(* Logix 5000 project; controller Generic 1768-L43 rev 16.2; software revision 15.01; part 5 of 10 *)
(* tags used below, declared in another part *)
   EL_CTRL_1 : UDT_AxisHistory_CTRL;
   EL_CTRL_2 : UDT_AxisHistory_CTRL;
   EL_CTRL_3 : UDT_AxisHistory_CTRL;
   EL_CTRL_4 : UDT_AxisHistory_CTRL;
   EL_CTRL_5 : UDT_AxisHistory_CTRL;
   EL_CTRL_6 : UDT_AxisHistory_CTRL;
   EL_CTRL_7 : UDT_AxisHistory_CTRL;
   EL_CTRL_8 : UDT_AxisHistory_CTRL;
   EL_SaveSEQ : DINT;
   EventINDEX : DINT;
   EventLog_N1 : UDT_AxisHistory_DLM[51];
   EventLog_N2 : UDT_AxisHistory_DLM[51];
   EventLog_N3 : UDT_AxisHistory_DLM[51];
   EventLog_N4 : UDT_AxisHistory_DLM[51];
   EventLog_N5 : UDT_AxisHistory_DLM[51];
   EventLog_N6 : UDT_AxisHistory_DLM[51];
   EventLog_N7 : UDT_AxisHistory_DLM[51];
   EventLog_N8 : UDT_AxisHistory_DLM[51];
   GUI_DataDisplay : UDT_AxisHistory_DLM;
   GUI_DataLogModel : UDT_AxisHistory_DLM;
   GUI_EventLogSaving : BOOL;
   GUI_IndexSelect : DINT;
   GUI_NodeSelect : DINT;
   GUI_SaveEventLog : BOOL;
   LogLength : DINT;
   PowerUP_TMR : TIMER;
   Axis_00_Data : UDT_Axis_Data;
   Axis_00_Status : UDT_Axis_Status;
   AXIS_01 : AXIS_SERVO_DRIVE;
   Axis_01_Data : UDT_Axis_Data;
   Axis_01_Status : UDT_Axis_Status;
   AXIS_02 : AXIS_SERVO_DRIVE;
   Axis_02_Data : UDT_Axis_Data;
   Axis_02_Status : UDT_Axis_Status;
   AXIS_03 : AXIS_SERVO_DRIVE;
   Axis_03_Data : UDT_Axis_Data;
   Axis_03_Status : UDT_Axis_Status;
   AXIS_04 : AXIS_SERVO_DRIVE;
   Axis_04_Data : UDT_Axis_Data;
   Axis_04_Status : UDT_Axis_Status;
   C_pi : REAL;
   GenericMachine_COND : UDT_Machine_COND;
   MASK : DINT;
(* AXIS_EventLog, continued *)

ROUTINE R20_HMI_EventLog   (* ladder *)
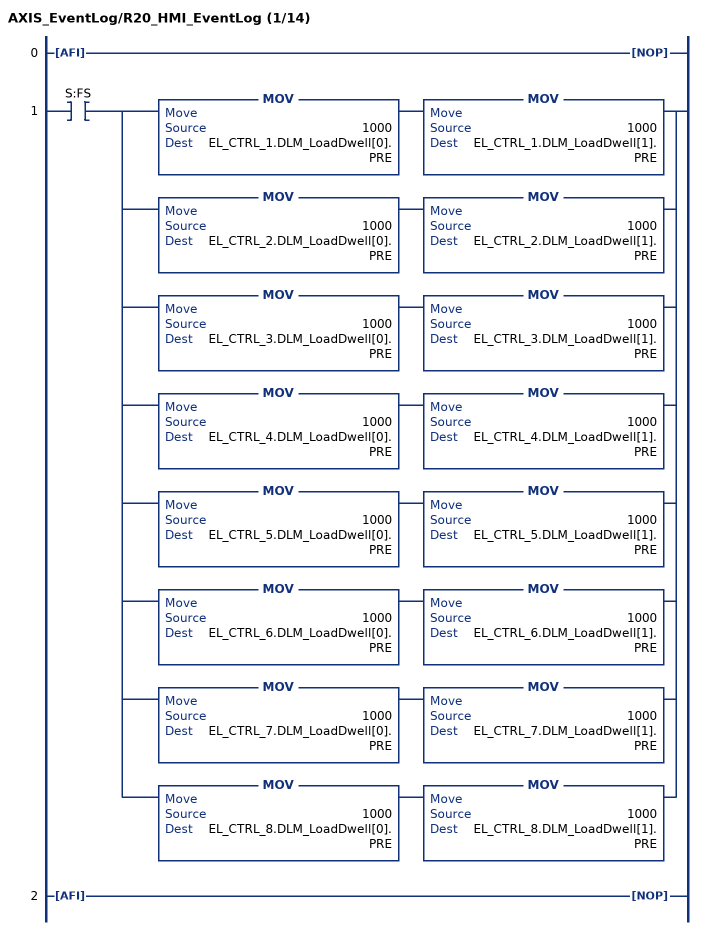
   0: AFI()NOP();
   1: XIC(S:FS)[MOV(1000,EL_CTRL_1.DLM_LoadDwell[0].PRE) MOV(1000,EL_CTRL_1.DLM_LoadDwell[1].PRE) ,MOV(1000,EL_CTRL_2.DLM_LoadDwell[0].PRE) MOV(1000,EL_CTRL_2.DLM_LoadDwell[1].PRE) ,MOV(1000,EL_CTRL_3.DLM_LoadDwell[0].PRE) MOV(1000,EL_CTRL_3.DLM_LoadDwell[1].PRE) ,MOV(1000,EL_CTRL_4.DLM_LoadDwell[0].PRE) MOV(1000,EL_CTRL_4.DLM_LoadDwell[1].PRE) ,MOV(1000,EL_CTRL_5.DLM_LoadDwell[0].PRE) MOV(1000,EL_CTRL_5.DLM_LoadDwell[1].PRE) ,MOV(1000,EL_CTRL_6.DLM_LoadDwell[0].PRE) MOV(1000,EL_CTRL_6.DLM_LoadDwell[1].PRE) ,MOV(1000,EL_CTRL_7.DLM_LoadDwell[0].PRE) MOV(1000,EL_CTRL_7.DLM_LoadDwell[1].PRE) ,MOV(1000,EL_CTRL_8.DLM_LoadDwell[0].PRE) MOV(1000,EL_CTRL_8.DLM_LoadDwell[1].PRE) ];
   2: AFI()NOP();
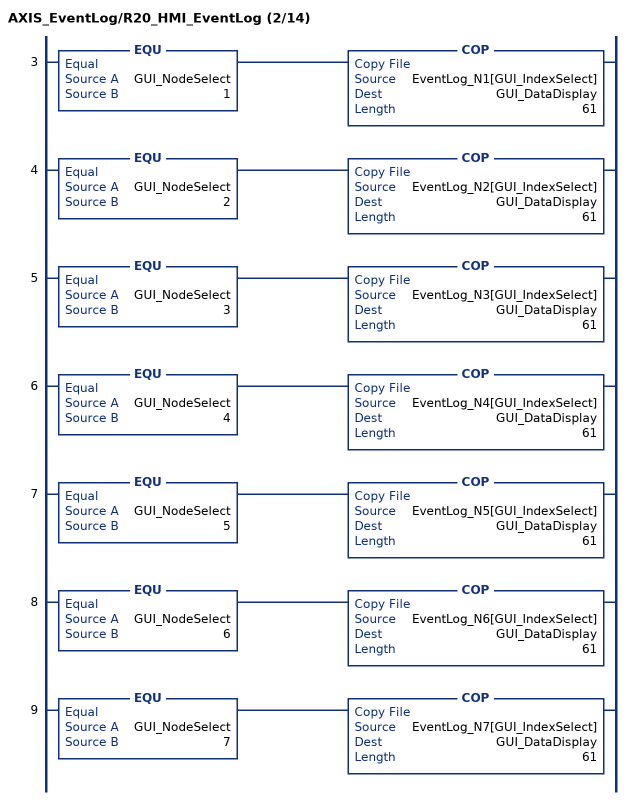
   3: EQU(GUI_NodeSelect,1)COP(EventLog_N1[GUI_IndexSelect],GUI_DataDisplay,61);
   4: EQU(GUI_NodeSelect,2)COP(EventLog_N2[GUI_IndexSelect],GUI_DataDisplay,61);
   5: EQU(GUI_NodeSelect,3)COP(EventLog_N3[GUI_IndexSelect],GUI_DataDisplay,61);
   6: EQU(GUI_NodeSelect,4)COP(EventLog_N4[GUI_IndexSelect],GUI_DataDisplay,61);
   7: EQU(GUI_NodeSelect,5)COP(EventLog_N5[GUI_IndexSelect],GUI_DataDisplay,61);
   8: EQU(GUI_NodeSelect,6)COP(EventLog_N6[GUI_IndexSelect],GUI_DataDisplay,61);
   9: EQU(GUI_NodeSelect,7)COP(EventLog_N7[GUI_IndexSelect],GUI_DataDisplay,61);
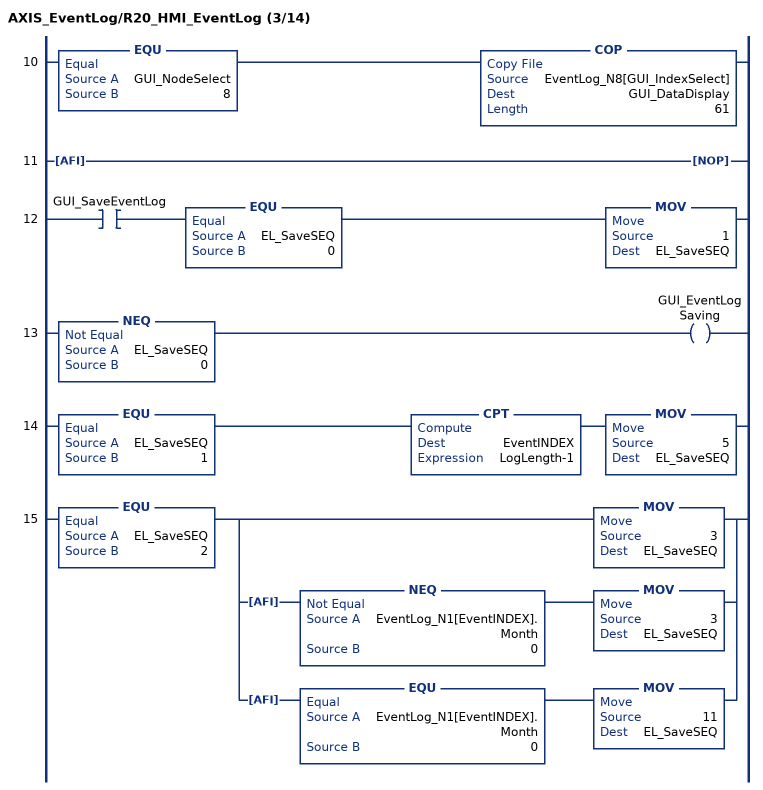
   10: EQU(GUI_NodeSelect,8)COP(EventLog_N8[GUI_IndexSelect],GUI_DataDisplay,61);
   11: AFI()NOP();
   12: XIC(GUI_SaveEventLog)EQU(EL_SaveSEQ,0)MOV(1,EL_SaveSEQ);
   13: NEQ(EL_SaveSEQ,0)OTE(GUI_EventLogSaving);
   14: EQU(EL_SaveSEQ,1)CPT(EventINDEX,LogLength-1)MOV(5,EL_SaveSEQ);
   15: EQU(EL_SaveSEQ,2)[MOV(3,EL_SaveSEQ) ,AFI() NEQ(EventLog_N1[EventINDEX].Month,0) MOV(3,EL_SaveSEQ) ,AFI() EQU(EventLog_N1[EventINDEX].Month,0) MOV(11,EL_SaveSEQ) ];
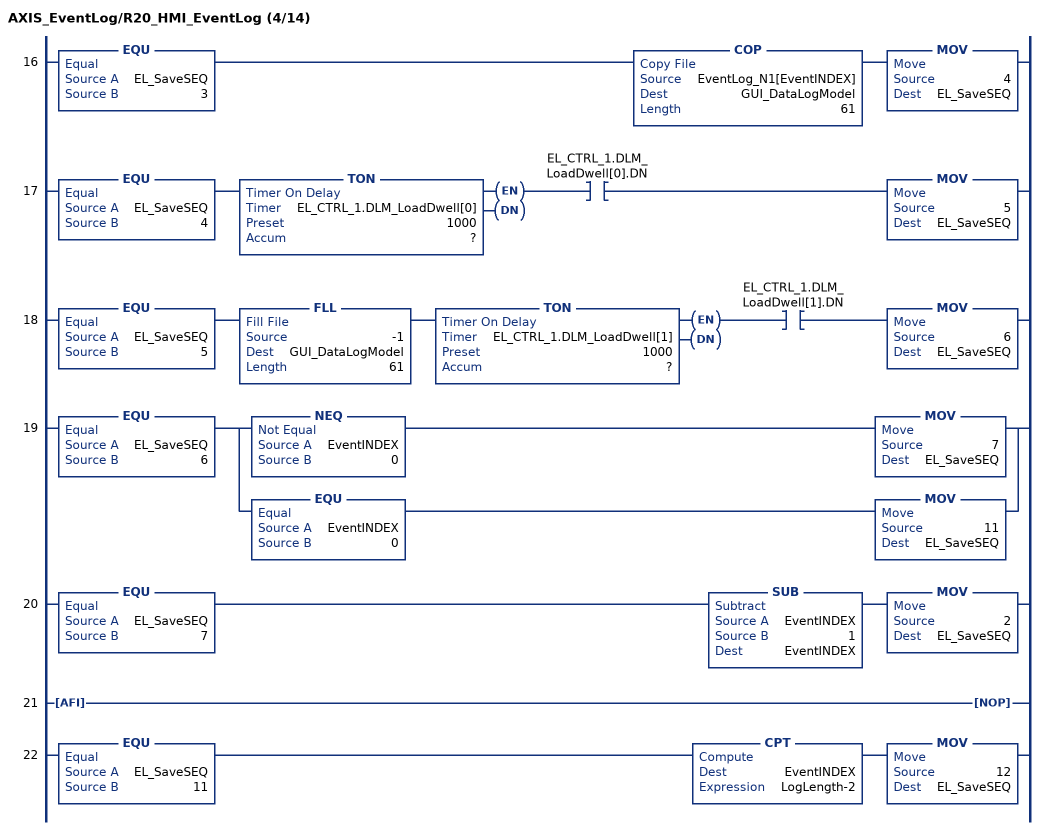
   16: EQU(EL_SaveSEQ,3)COP(EventLog_N1[EventINDEX],GUI_DataLogModel,61)MOV(4,EL_SaveSEQ);
   17: EQU(EL_SaveSEQ,4)TON(EL_CTRL_1.DLM_LoadDwell[0],?,?)XIC(EL_CTRL_1.DLM_LoadDwell[0].DN)MOV(5,EL_SaveSEQ);
   18: EQU(EL_SaveSEQ,5)FLL(-1,GUI_DataLogModel,61)TON(EL_CTRL_1.DLM_LoadDwell[1],?,?)XIC(EL_CTRL_1.DLM_LoadDwell[1].DN)MOV(6,EL_SaveSEQ);
   19: EQU(EL_SaveSEQ,6)[NEQ(EventINDEX,0) MOV(7,EL_SaveSEQ) ,EQU(EventINDEX,0) MOV(11,EL_SaveSEQ) ];
   20: EQU(EL_SaveSEQ,7)SUB(EventINDEX,1,EventINDEX)MOV(2,EL_SaveSEQ);
   21: AFI()NOP();
   22: EQU(EL_SaveSEQ,11)CPT(EventINDEX,LogLength-2)MOV(12,EL_SaveSEQ);
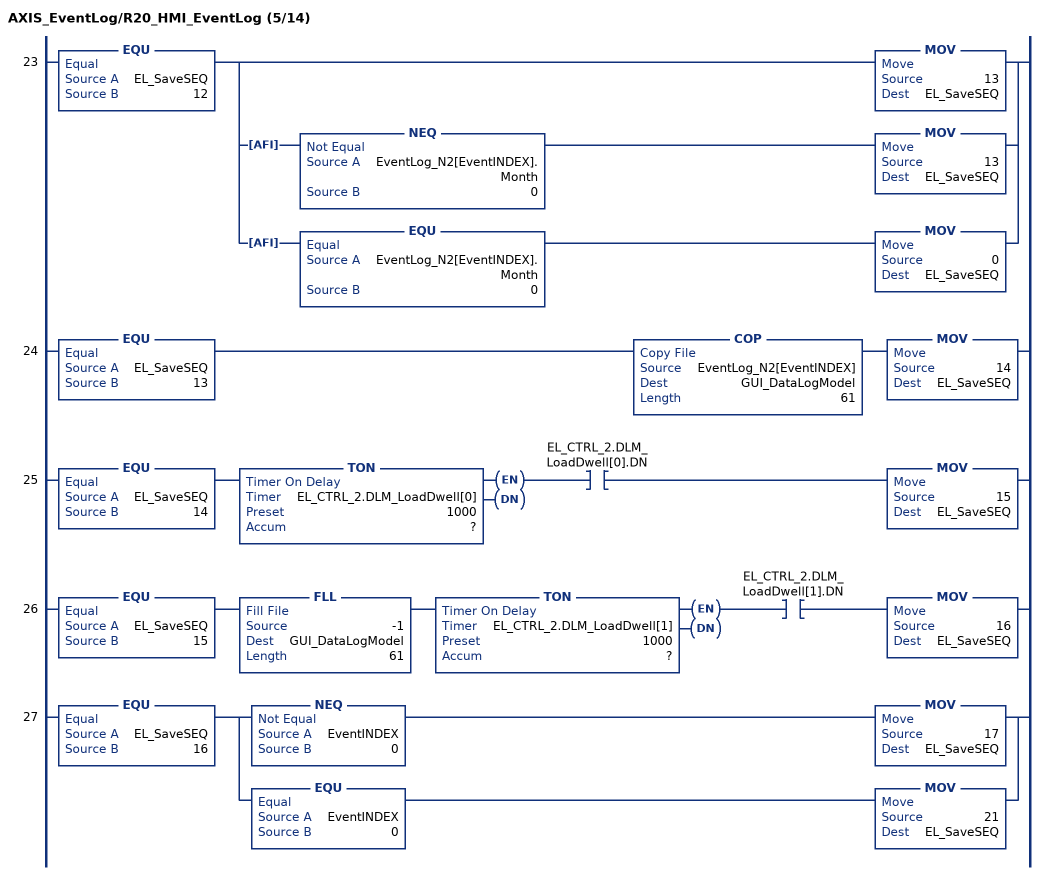
   23: EQU(EL_SaveSEQ,12)[MOV(13,EL_SaveSEQ) ,AFI() NEQ(EventLog_N2[EventINDEX].Month,0) MOV(13,EL_SaveSEQ) ,AFI() EQU(EventLog_N2[EventINDEX].Month,0) MOV(0,EL_SaveSEQ) ];
   24: EQU(EL_SaveSEQ,13)COP(EventLog_N2[EventINDEX],GUI_DataLogModel,61)MOV(14,EL_SaveSEQ);
   25: EQU(EL_SaveSEQ,14)TON(EL_CTRL_2.DLM_LoadDwell[0],?,?)XIC(EL_CTRL_2.DLM_LoadDwell[0].DN)MOV(15,EL_SaveSEQ);
   26: EQU(EL_SaveSEQ,15)FLL(-1,GUI_DataLogModel,61)TON(EL_CTRL_2.DLM_LoadDwell[1],?,?)XIC(EL_CTRL_2.DLM_LoadDwell[1].DN)MOV(16,EL_SaveSEQ);
   27: EQU(EL_SaveSEQ,16)[NEQ(EventINDEX,0) MOV(17,EL_SaveSEQ) ,EQU(EventINDEX,0) MOV(21,EL_SaveSEQ) ];
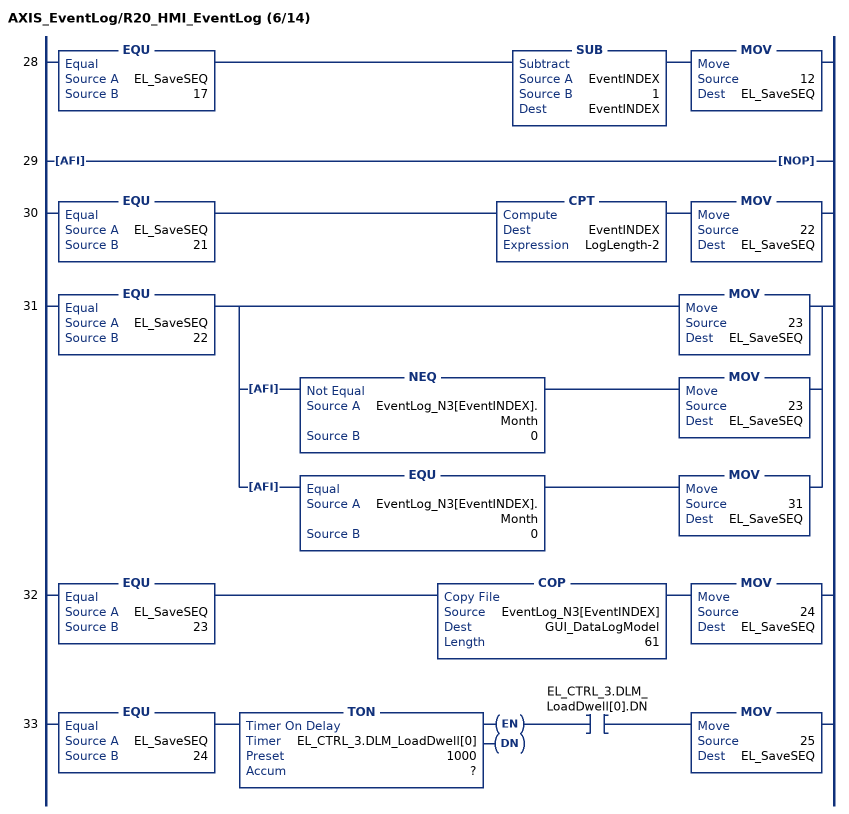
   28: EQU(EL_SaveSEQ,17)SUB(EventINDEX,1,EventINDEX)MOV(12,EL_SaveSEQ);
   29: AFI()NOP();
   30: EQU(EL_SaveSEQ,21)CPT(EventINDEX,LogLength-2)MOV(22,EL_SaveSEQ);
   31: EQU(EL_SaveSEQ,22)[MOV(23,EL_SaveSEQ) ,AFI() NEQ(EventLog_N3[EventINDEX].Month,0) MOV(23,EL_SaveSEQ) ,AFI() EQU(EventLog_N3[EventINDEX].Month,0) MOV(31,EL_SaveSEQ) ];
   32: EQU(EL_SaveSEQ,23)COP(EventLog_N3[EventINDEX],GUI_DataLogModel,61)MOV(24,EL_SaveSEQ);
   33: EQU(EL_SaveSEQ,24)TON(EL_CTRL_3.DLM_LoadDwell[0],?,?)XIC(EL_CTRL_3.DLM_LoadDwell[0].DN)MOV(25,EL_SaveSEQ);
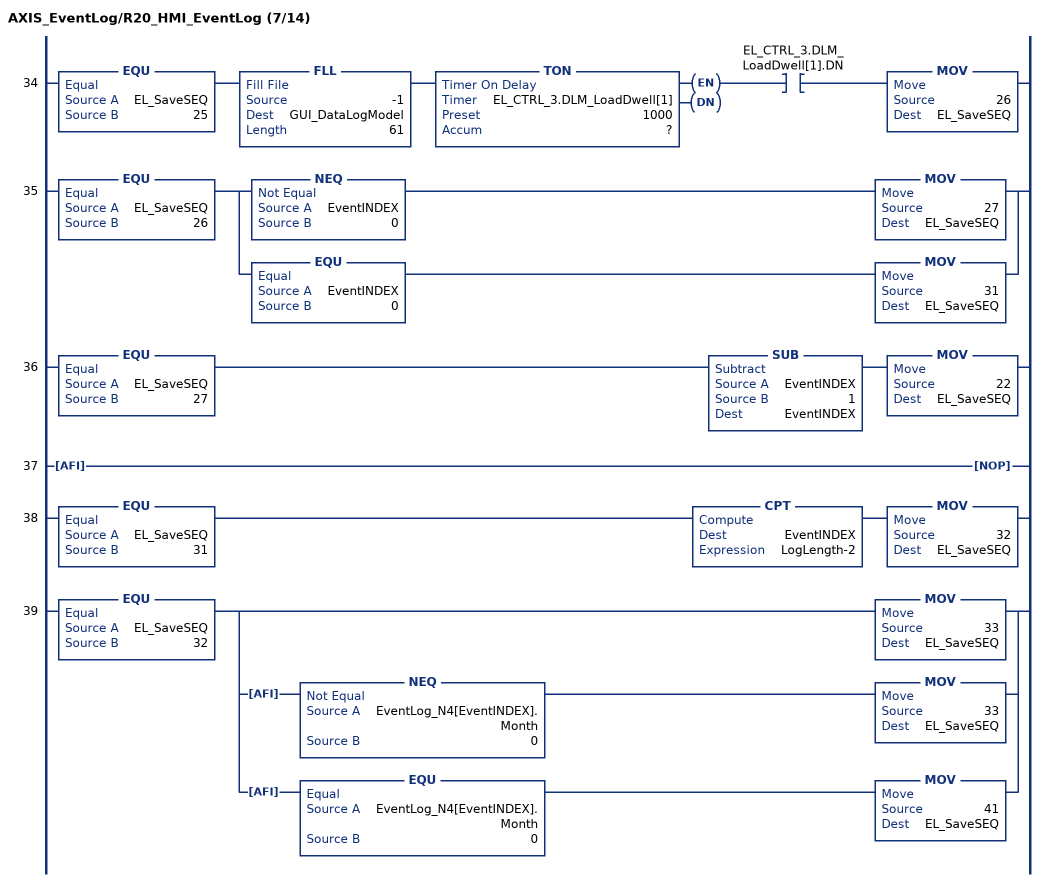
   34: EQU(EL_SaveSEQ,25)FLL(-1,GUI_DataLogModel,61)TON(EL_CTRL_3.DLM_LoadDwell[1],?,?)XIC(EL_CTRL_3.DLM_LoadDwell[1].DN)MOV(26,EL_SaveSEQ);
   35: EQU(EL_SaveSEQ,26)[NEQ(EventINDEX,0) MOV(27,EL_SaveSEQ) ,EQU(EventINDEX,0) MOV(31,EL_SaveSEQ) ];
   36: EQU(EL_SaveSEQ,27)SUB(EventINDEX,1,EventINDEX)MOV(22,EL_SaveSEQ);
   37: AFI()NOP();
   38: EQU(EL_SaveSEQ,31)CPT(EventINDEX,LogLength-2)MOV(32,EL_SaveSEQ);
   39: EQU(EL_SaveSEQ,32)[MOV(33,EL_SaveSEQ) ,AFI() NEQ(EventLog_N4[EventINDEX].Month,0) MOV(33,EL_SaveSEQ) ,AFI() EQU(EventLog_N4[EventINDEX].Month,0) MOV(41,EL_SaveSEQ) ];
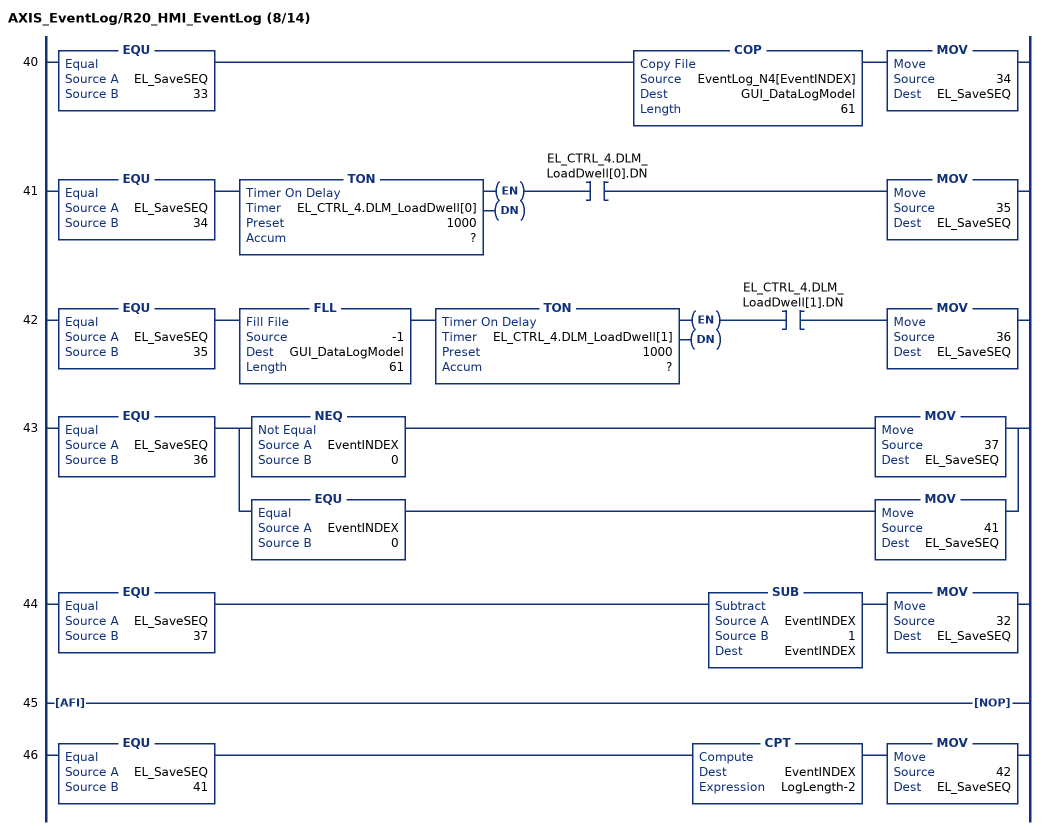
   40: EQU(EL_SaveSEQ,33)COP(EventLog_N4[EventINDEX],GUI_DataLogModel,61)MOV(34,EL_SaveSEQ);
   41: EQU(EL_SaveSEQ,34)TON(EL_CTRL_4.DLM_LoadDwell[0],?,?)XIC(EL_CTRL_4.DLM_LoadDwell[0].DN)MOV(35,EL_SaveSEQ);
   42: EQU(EL_SaveSEQ,35)FLL(-1,GUI_DataLogModel,61)TON(EL_CTRL_4.DLM_LoadDwell[1],?,?)XIC(EL_CTRL_4.DLM_LoadDwell[1].DN)MOV(36,EL_SaveSEQ);
   43: EQU(EL_SaveSEQ,36)[NEQ(EventINDEX,0) MOV(37,EL_SaveSEQ) ,EQU(EventINDEX,0) MOV(41,EL_SaveSEQ) ];
   44: EQU(EL_SaveSEQ,37)SUB(EventINDEX,1,EventINDEX)MOV(32,EL_SaveSEQ);
   45: AFI()NOP();
   46: EQU(EL_SaveSEQ,41)CPT(EventINDEX,LogLength-2)MOV(42,EL_SaveSEQ);
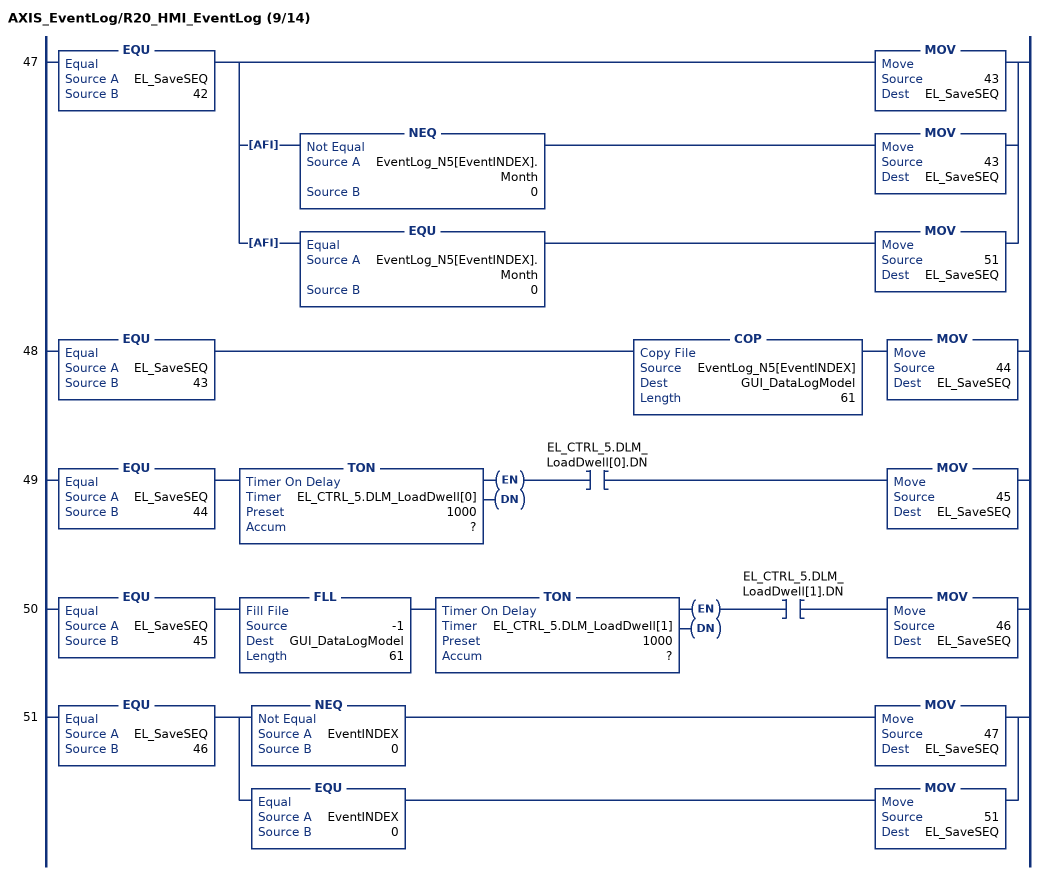
   47: EQU(EL_SaveSEQ,42)[MOV(43,EL_SaveSEQ) ,AFI() NEQ(EventLog_N5[EventINDEX].Month,0) MOV(43,EL_SaveSEQ) ,AFI() EQU(EventLog_N5[EventINDEX].Month,0) MOV(51,EL_SaveSEQ) ];
   48: EQU(EL_SaveSEQ,43)COP(EventLog_N5[EventINDEX],GUI_DataLogModel,61)MOV(44,EL_SaveSEQ);
   49: EQU(EL_SaveSEQ,44)TON(EL_CTRL_5.DLM_LoadDwell[0],?,?)XIC(EL_CTRL_5.DLM_LoadDwell[0].DN)MOV(45,EL_SaveSEQ);
   50: EQU(EL_SaveSEQ,45)FLL(-1,GUI_DataLogModel,61)TON(EL_CTRL_5.DLM_LoadDwell[1],?,?)XIC(EL_CTRL_5.DLM_LoadDwell[1].DN)MOV(46,EL_SaveSEQ);
   51: EQU(EL_SaveSEQ,46)[NEQ(EventINDEX,0) MOV(47,EL_SaveSEQ) ,EQU(EventINDEX,0) MOV(51,EL_SaveSEQ) ];
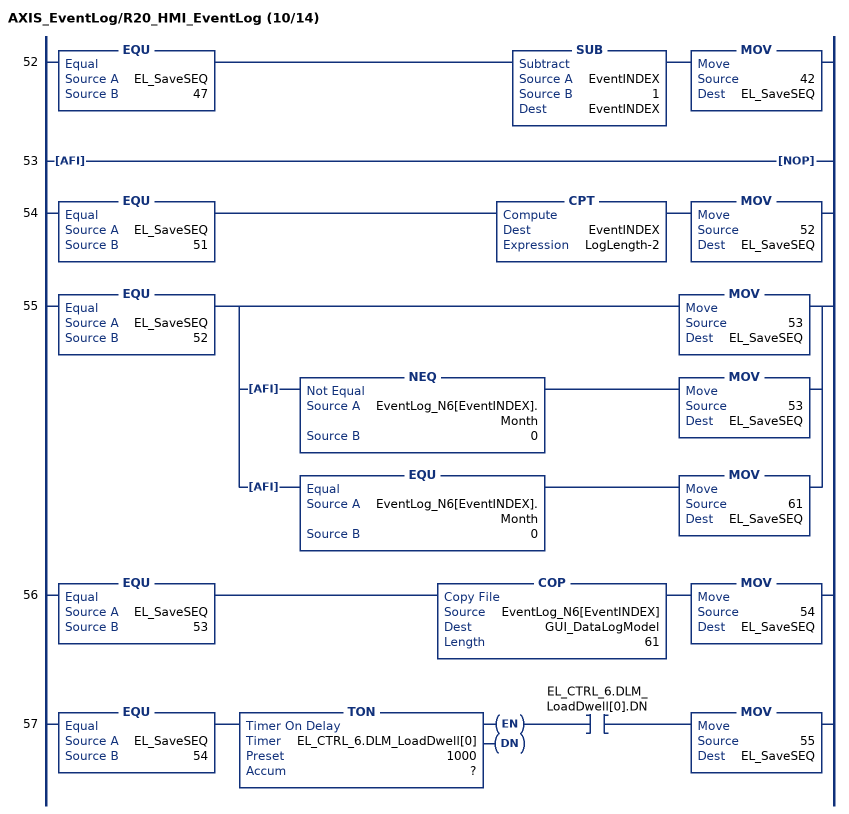
   52: EQU(EL_SaveSEQ,47)SUB(EventINDEX,1,EventINDEX)MOV(42,EL_SaveSEQ);
   53: AFI()NOP();
   54: EQU(EL_SaveSEQ,51)CPT(EventINDEX,LogLength-2)MOV(52,EL_SaveSEQ);
   55: EQU(EL_SaveSEQ,52)[MOV(53,EL_SaveSEQ) ,AFI() NEQ(EventLog_N6[EventINDEX].Month,0) MOV(53,EL_SaveSEQ) ,AFI() EQU(EventLog_N6[EventINDEX].Month,0) MOV(61,EL_SaveSEQ) ];
   56: EQU(EL_SaveSEQ,53)COP(EventLog_N6[EventINDEX],GUI_DataLogModel,61)MOV(54,EL_SaveSEQ);
   57: EQU(EL_SaveSEQ,54)TON(EL_CTRL_6.DLM_LoadDwell[0],?,?)XIC(EL_CTRL_6.DLM_LoadDwell[0].DN)MOV(55,EL_SaveSEQ);
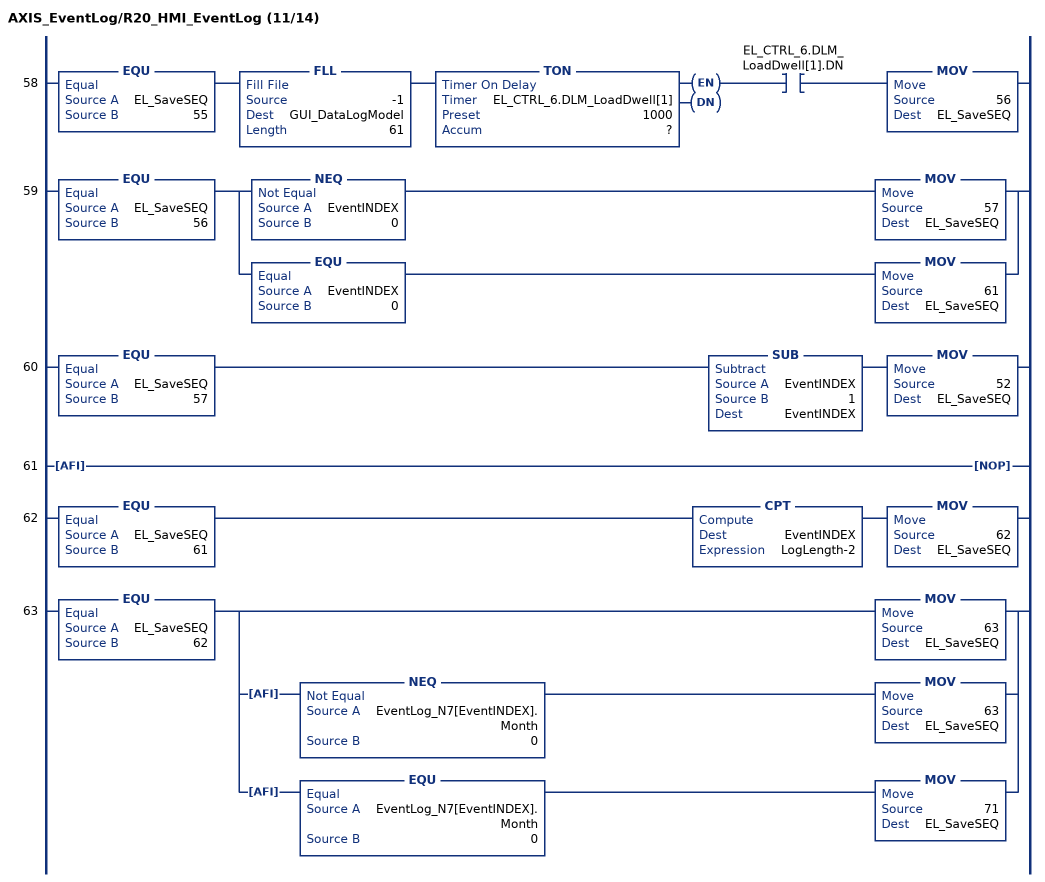
   58: EQU(EL_SaveSEQ,55)FLL(-1,GUI_DataLogModel,61)TON(EL_CTRL_6.DLM_LoadDwell[1],?,?)XIC(EL_CTRL_6.DLM_LoadDwell[1].DN)MOV(56,EL_SaveSEQ);
   59: EQU(EL_SaveSEQ,56)[NEQ(EventINDEX,0) MOV(57,EL_SaveSEQ) ,EQU(EventINDEX,0) MOV(61,EL_SaveSEQ) ];
   60: EQU(EL_SaveSEQ,57)SUB(EventINDEX,1,EventINDEX)MOV(52,EL_SaveSEQ);
   61: AFI()NOP();
   62: EQU(EL_SaveSEQ,61)CPT(EventINDEX,LogLength-2)MOV(62,EL_SaveSEQ);
   63: EQU(EL_SaveSEQ,62)[MOV(63,EL_SaveSEQ) ,AFI() NEQ(EventLog_N7[EventINDEX].Month,0) MOV(63,EL_SaveSEQ) ,AFI() EQU(EventLog_N7[EventINDEX].Month,0) MOV(71,EL_SaveSEQ) ];
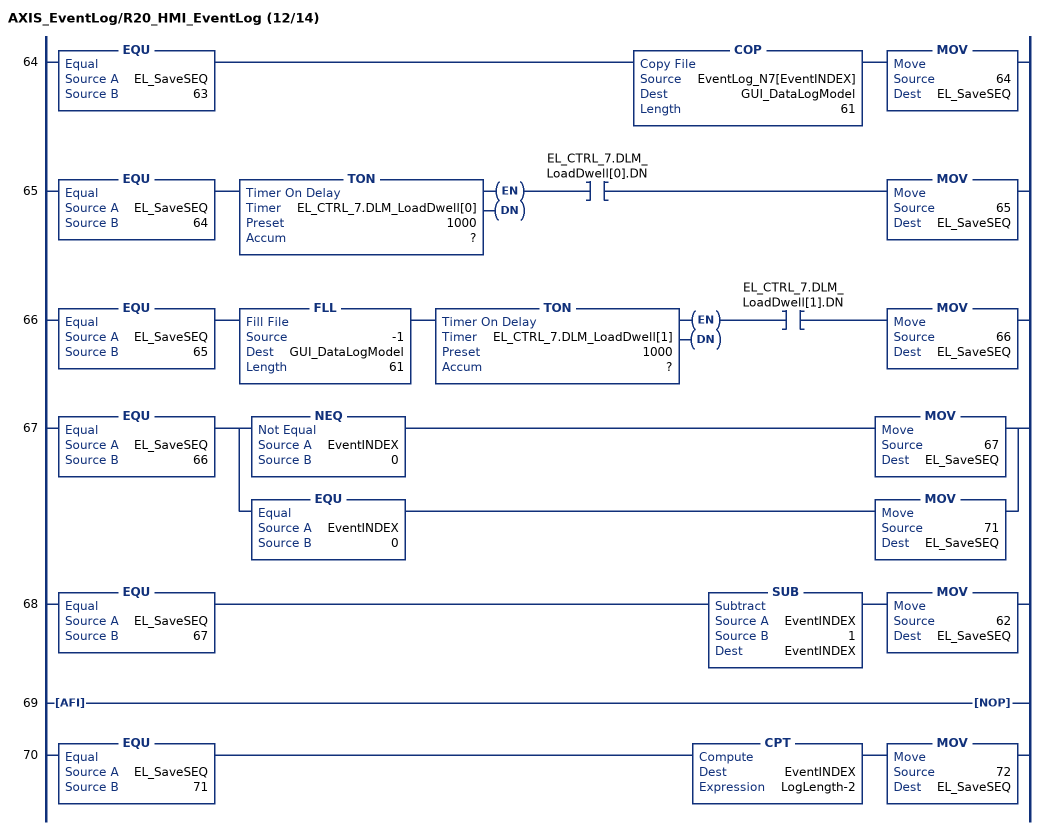
   64: EQU(EL_SaveSEQ,63)COP(EventLog_N7[EventINDEX],GUI_DataLogModel,61)MOV(64,EL_SaveSEQ);
   65: EQU(EL_SaveSEQ,64)TON(EL_CTRL_7.DLM_LoadDwell[0],?,?)XIC(EL_CTRL_7.DLM_LoadDwell[0].DN)MOV(65,EL_SaveSEQ);
   66: EQU(EL_SaveSEQ,65)FLL(-1,GUI_DataLogModel,61)TON(EL_CTRL_7.DLM_LoadDwell[1],?,?)XIC(EL_CTRL_7.DLM_LoadDwell[1].DN)MOV(66,EL_SaveSEQ);
   67: EQU(EL_SaveSEQ,66)[NEQ(EventINDEX,0) MOV(67,EL_SaveSEQ) ,EQU(EventINDEX,0) MOV(71,EL_SaveSEQ) ];
   68: EQU(EL_SaveSEQ,67)SUB(EventINDEX,1,EventINDEX)MOV(62,EL_SaveSEQ);
   69: AFI()NOP();
   70: EQU(EL_SaveSEQ,71)CPT(EventINDEX,LogLength-2)MOV(72,EL_SaveSEQ);
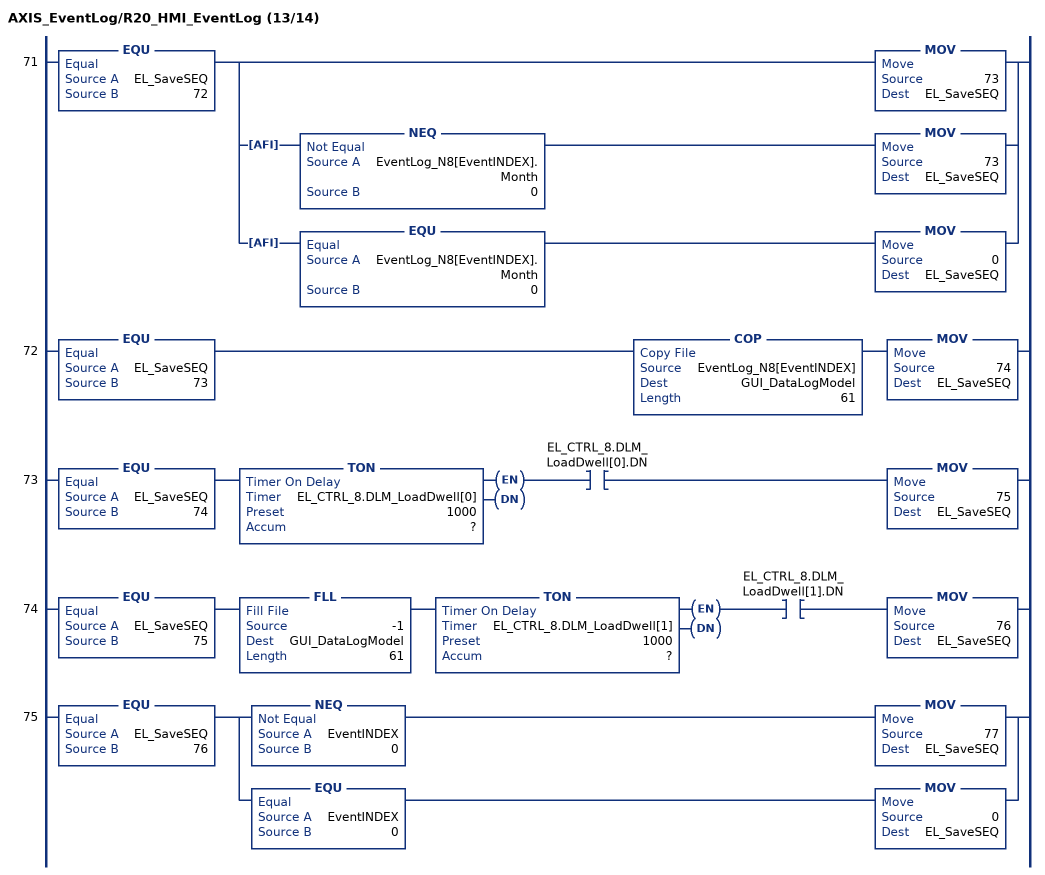
   71: EQU(EL_SaveSEQ,72)[MOV(73,EL_SaveSEQ) ,AFI() NEQ(EventLog_N8[EventINDEX].Month,0) MOV(73,EL_SaveSEQ) ,AFI() EQU(EventLog_N8[EventINDEX].Month,0) MOV(0,EL_SaveSEQ) ];
   72: EQU(EL_SaveSEQ,73)COP(EventLog_N8[EventINDEX],GUI_DataLogModel,61)MOV(74,EL_SaveSEQ);
   73: EQU(EL_SaveSEQ,74)TON(EL_CTRL_8.DLM_LoadDwell[0],?,?)XIC(EL_CTRL_8.DLM_LoadDwell[0].DN)MOV(75,EL_SaveSEQ);
   74: EQU(EL_SaveSEQ,75)FLL(-1,GUI_DataLogModel,61)TON(EL_CTRL_8.DLM_LoadDwell[1],?,?)XIC(EL_CTRL_8.DLM_LoadDwell[1].DN)MOV(76,EL_SaveSEQ);
   75: EQU(EL_SaveSEQ,76)[NEQ(EventINDEX,0) MOV(77,EL_SaveSEQ) ,EQU(EventINDEX,0) MOV(0,EL_SaveSEQ) ];
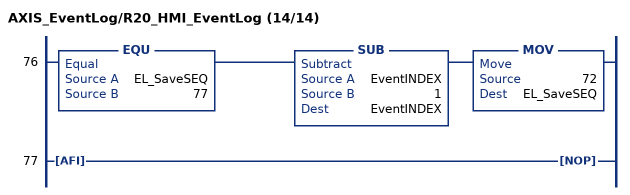
   76: EQU(EL_SaveSEQ,77)SUB(EventINDEX,1,EventINDEX)MOV(72,EL_SaveSEQ);
   77: AFI()NOP();
END_ROUTINE
END_PROGRAM

PROGRAM P00_Control   (* main routine R00_MainDispatch *)
VAR
   R04_OTE : DINT;
END_VAR

ROUTINE R00_MainDispatch   (* ladder *)
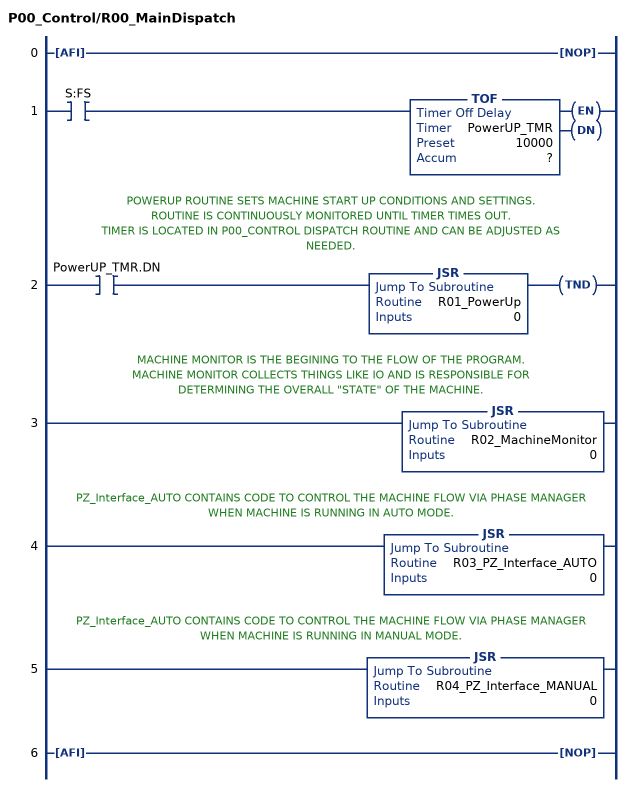
   0: AFI()NOP();
   1: XIC(S:FS)TOF(PowerUP_TMR,?,?);
   // POWERUP ROUTINE SETS MACHINE START UP CONDITIONS AND SETTINGS.
   // ROUTINE IS CONTINUOUSLY MONITORED UNTIL TIMER TIMES OUT.
   // TIMER IS LOCATED IN P00_CONTROL DISPATCH ROUTINE AND CAN BE ADJUSTED AS NEEDED.
   2: XIC(PowerUP_TMR.DN)JSR(R01_PowerUp,0)TND();
   // MACHINE MONITOR IS THE BEGINING TO THE FLOW OF THE PROGRAM.
   // MACHINE MONITOR COLLECTS THINGS LIKE IO AND IS RESPONSIBLE FOR
   // DETERMINING THE OVERALL "STATE" OF THE MACHINE.
   3: JSR(R02_MachineMonitor,0);
   // PZ_Interface_AUTO CONTAINS CODE TO CONTROL THE MACHINE FLOW VIA PHASE MANAGER
   //  WHEN MACHINE IS RUNNING IN AUTO MODE.
   4: JSR(R03_PZ_Interface_AUTO,0);
   // PZ_Interface_AUTO CONTAINS CODE TO CONTROL THE MACHINE FLOW VIA PHASE MANAGER
   //  WHEN MACHINE IS RUNNING IN MANUAL MODE.
   5: JSR(R04_PZ_Interface_MANUAL,0);
   6: AFI()NOP();
END_ROUTINE

ROUTINE R01_PowerUp   (* ladder *)
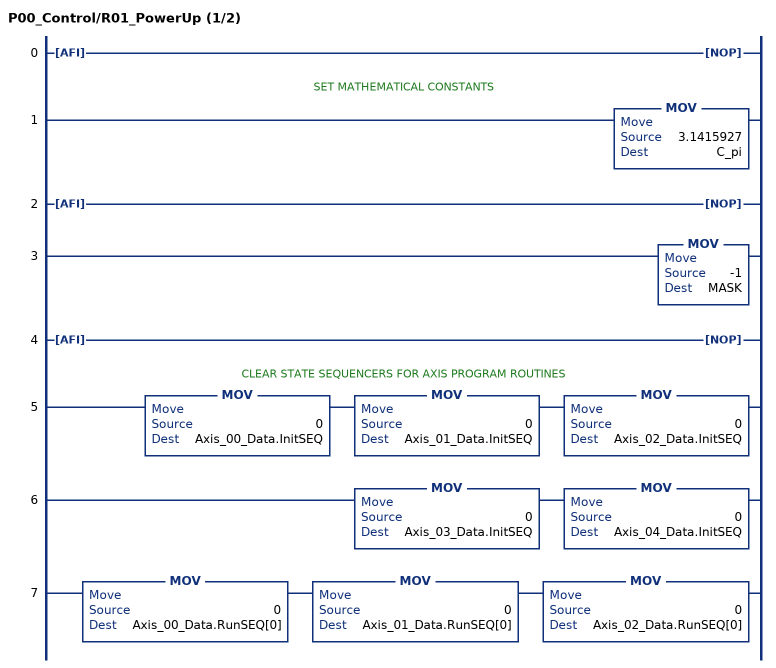
   0: AFI()NOP();
   // SET MATHEMATICAL CONSTANTS
   1: MOV(3.1415927,C_pi);
   2: AFI()NOP();
   3: MOV(-1,MASK);
   4: AFI()NOP();
   // CLEAR STATE SEQUENCERS FOR AXIS PROGRAM ROUTINES
   5: MOV(0,Axis_00_Data.InitSEQ)MOV(0,Axis_01_Data.InitSEQ)MOV(0,Axis_02_Data.InitSEQ);
   6: MOV(0,Axis_03_Data.InitSEQ)MOV(0,Axis_04_Data.InitSEQ);
   7: MOV(0,Axis_00_Data.RunSEQ[0])MOV(0,Axis_01_Data.RunSEQ[0])MOV(0,Axis_02_Data.RunSEQ[0]);
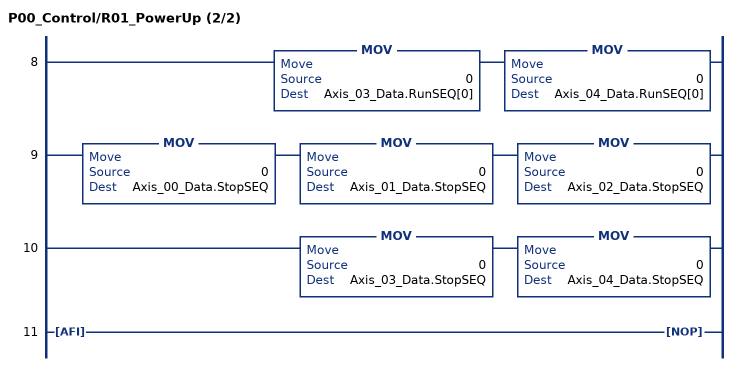
   8: MOV(0,Axis_03_Data.RunSEQ[0])MOV(0,Axis_04_Data.RunSEQ[0]);
   9: MOV(0,Axis_00_Data.StopSEQ)MOV(0,Axis_01_Data.StopSEQ)MOV(0,Axis_02_Data.StopSEQ);
   10: MOV(0,Axis_03_Data.StopSEQ)MOV(0,Axis_04_Data.StopSEQ);
   11: AFI()NOP();
END_ROUTINE

ROUTINE R02_MachineMonitor   (* ladder *)
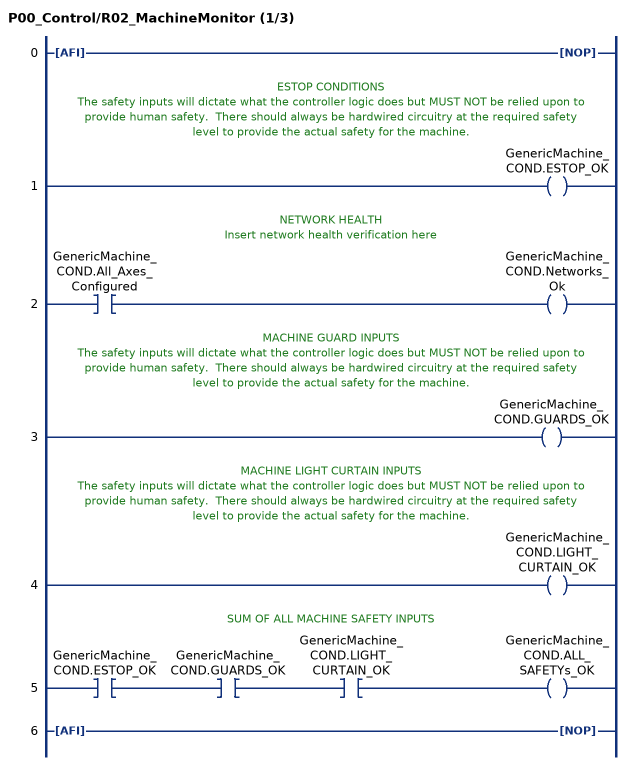
   0: AFI()NOP();
   // ESTOP CONDITIONS
   // The safety inputs will dictate what the controller logic does but MUST NOT be relied upon to provide human safety.  There should always be hardwired circuitry at the required safety level to provide the actual safety for the machine.
   1: OTE(GenericMachine_COND.ESTOP_OK);
   // NETWORK HEALTH
   // Insert network health verification here
   2: XIC(GenericMachine_COND.All_Axes_Configured)OTE(GenericMachine_COND.Networks_Ok);
   // MACHINE GUARD INPUTS
   // The safety inputs will dictate what the controller logic does but MUST NOT be relied upon to provide human safety.  There should always be hardwired circuitry at the required safety level to provide the actual safety for the machine.
   3: OTE(GenericMachine_COND.GUARDS_OK);
   // MACHINE LIGHT CURTAIN INPUTS
   // The safety inputs will dictate what the controller logic does but MUST NOT be relied upon to provide human safety.  There should always be hardwired circuitry at the required safety level to provide the actual safety for the machine.
   4: OTE(GenericMachine_COND.LIGHT_CURTAIN_OK);
   // SUM OF ALL MACHINE SAFETY INPUTS
   5: XIC(GenericMachine_COND.ESTOP_OK)XIC(GenericMachine_COND.GUARDS_OK)XIC(GenericMachine_COND.LIGHT_CURTAIN_OK)OTE(GenericMachine_COND.ALL_SAFETYs_OK);
   6: AFI()NOP();
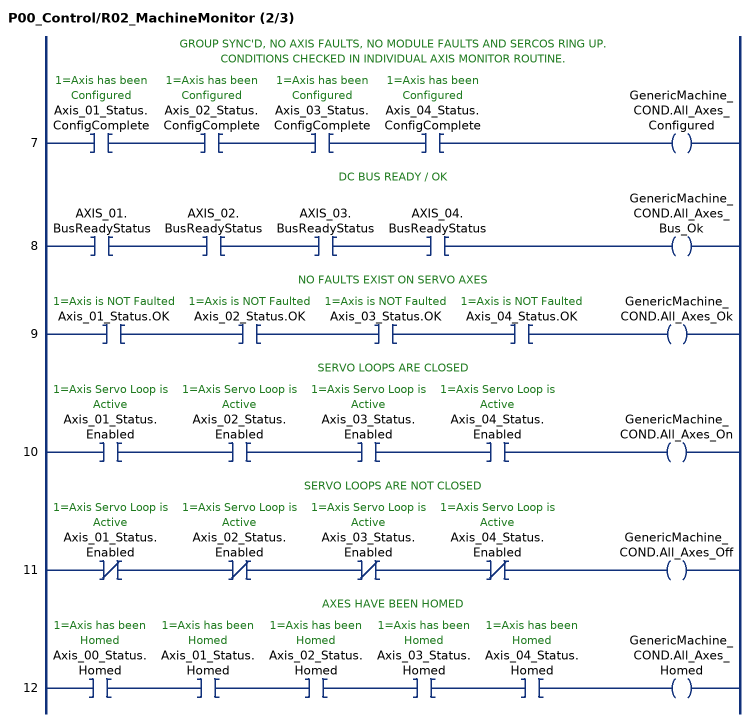
   // GROUP SYNC'D, NO AXIS FAULTS, NO MODULE FAULTS AND SERCOS RING UP.
   // CONDITIONS CHECKED IN INDIVIDUAL AXIS MONITOR ROUTINE.
   7: XIC(Axis_01_Status.ConfigComplete)XIC(Axis_02_Status.ConfigComplete)XIC(Axis_03_Status.ConfigComplete)XIC(Axis_04_Status.ConfigComplete)OTE(GenericMachine_COND.All_Axes_Configured);
   // DC BUS READY / OK
   8: XIC(AXIS_01.BusReadyStatus)XIC(AXIS_02.BusReadyStatus)XIC(AXIS_03.BusReadyStatus)XIC(AXIS_04.BusReadyStatus)OTE(GenericMachine_COND.All_Axes_Bus_Ok);
   // NO FAULTS EXIST ON SERVO AXES
   9: XIC(Axis_01_Status.OK)XIC(Axis_02_Status.OK)XIC(Axis_03_Status.OK)XIC(Axis_04_Status.OK)OTE(GenericMachine_COND.All_Axes_Ok);
   // SERVO LOOPS ARE CLOSED
   10: XIC(Axis_01_Status.Enabled)XIC(Axis_02_Status.Enabled)XIC(Axis_03_Status.Enabled)XIC(Axis_04_Status.Enabled)OTE(GenericMachine_COND.All_Axes_On);
   // SERVO LOOPS ARE NOT CLOSED
   11: XIO(Axis_01_Status.Enabled)XIO(Axis_02_Status.Enabled)XIO(Axis_03_Status.Enabled)XIO(Axis_04_Status.Enabled)OTE(GenericMachine_COND.All_Axes_Off);
   // AXES HAVE BEEN HOMED
   12: XIC(Axis_00_Status.Homed)XIC(Axis_01_Status.Homed)XIC(Axis_02_Status.Homed)XIC(Axis_03_Status.Homed)XIC(Axis_04_Status.Homed)OTE(GenericMachine_COND.All_Axes_Homed);
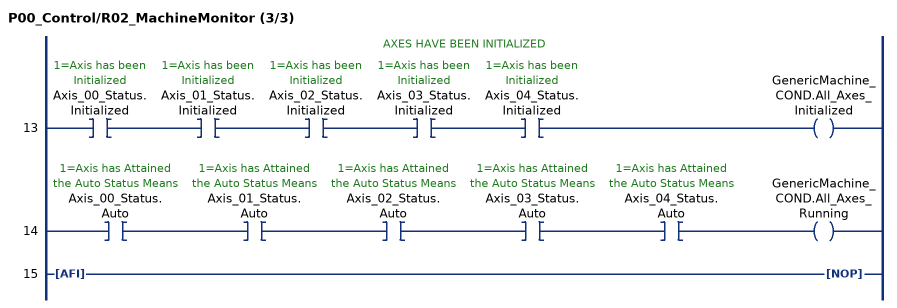
   // AXES HAVE BEEN INITIALIZED
   13: XIC(Axis_00_Status.Initialized)XIC(Axis_01_Status.Initialized)XIC(Axis_02_Status.Initialized)XIC(Axis_03_Status.Initialized)XIC(Axis_04_Status.Initialized)OTE(GenericMachine_COND.All_Axes_Initialized);
   14: XIC(Axis_00_Status.Auto)XIC(Axis_01_Status.Auto)XIC(Axis_02_Status.Auto)XIC(Axis_03_Status.Auto)XIC(Axis_04_Status.Auto)OTE(GenericMachine_COND.All_Axes_Running);
   15: AFI()NOP();
END_ROUTINE
